FUNCTION_BLOCK GET_AT_INDEX
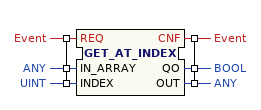
  EVENT_INPUT
    REQ WITH IN_ARRAY, INDEX;
  END_EVENT
  EVENT_OUTPUT
    CNF WITH QO, OUT;
  END_EVENT
  VAR_INPUT
    IN_ARRAY : ANY;
    INDEX : UINT;
  END_VAR
  VAR_OUTPUT
    QO : BOOL;
    OUT : ANY;
  END_VAR
END_FUNCTION_BLOCK
